DECL BOOL FraesAnford[10]
FraesAnford[1]=TRUE
FraesAnford[2]=TRUE
FraesAnford[3]=TRUE
FraesAnford[4]=FALSE
FraesAnford[5]=FALSE
FraesAnford[6]=FALSE
FraesAnford[7]=FALSE
FraesAnford[8]=FALSE
FraesAnford[9]=FALSE
FraesAnford[10]=FALSE
INT ERROR_PRG=0
;ENDFOLD
;FOLD USERSPOT_INPUTS_V4.xx
INT MAX_I_PS_MESSAGE=110
DECL I_MESSAGETYP PS_MESSAGE[110]
; EINGAENGE AM MODUL ZANGE 1
PS_MESSAGE[1]={I_NR 67,I_MSG_TXT[] "Stroemungswaechter Zange 1 E67 S42B                   "}
PS_MESSAGE[2]={I_NR 69,I_MSG_TXT[] "Vorhub Zange 1 hinten E69 B41YER                        "}
PS_MESSAGE[3]={I_NR 70,I_MSG_TXT[] "Schweisshub Zange 1 offen E70 B40YER                    "}
PS_MESSAGE[4]={I_NR 71,I_MSG_TXT[] "X-Vorhub Zange 1 vorne E71 B41YEV                       "}
PS_MESSAGE[5]={I_NR 72,I_MSG_TXT[] "Thermoschutz Trafo Zange 1 E72 B42TH                    "}
PS_MESSAGE[6]={I_NR 0,I_MSG_TXT[] " "}
PS_MESSAGE[7]={I_NR 0,I_MSG_TXT[] " "}
PS_MESSAGE[8]={I_NR 0,I_MSG_TXT[] " "}
PS_MESSAGE[9]={I_NR 0,I_MSG_TXT[] " "}

; EINGAENGE AM MODUL ZANGE 2
PS_MESSAGE[10]={I_NR 83,I_MSG_TXT[] "Stroemungswaechter Zange 2 E83 S12B                     "}
PS_MESSAGE[11]={I_NR 85,I_MSG_TXT[] "Vorhub Zange 2 hinten E85 B11YER                        "}
PS_MESSAGE[12]={I_NR 86,I_MSG_TXT[] "Schweisshub Zange 2 offen E86 B10YER                    "}
PS_MESSAGE[13]={I_NR 87,I_MSG_TXT[] "X-Vorhub Zange 2 vorne E87 B11YEV                       "}
PS_MESSAGE[14]={I_NR 88,I_MSG_TXT[] "Thermoschutz Trafo Zange 2 E88 B12TH                    "}
PS_MESSAGE[15]={I_NR 0,I_MSG_TXT[] " "}
PS_MESSAGE[16]={I_NR 0,I_MSG_TXT[] " "}
PS_MESSAGE[17]={I_NR 0,I_MSG_TXT[] " "}
PS_MESSAGE[18]={I_NR 0,I_MSG_TXT[] " "}


; EINGAENGE AM MODUL ZANGE 3
PS_MESSAGE[19]={I_NR 99,I_MSG_TXT[] "Stroemungswaechter Zange 3 E99 S22B                     "}
PS_MESSAGE[20]={I_NR 101,I_MSG_TXT[] "Vorhub Zange 3 hinten E101 B21YER                       "}
PS_MESSAGE[21]={I_NR 102,I_MSG_TXT[] "Schweisshub Zange 3 offen E102 B20YER                   "}
PS_MESSAGE[22]={I_NR 103,I_MSG_TXT[] "X-Vorhub Zange 3 vorne E103 B21YEV                      "}
PS_MESSAGE[23]={I_NR 104,I_MSG_TXT[] "Thermoschutz Trafo Zange 3 E104 B22TH                   "}
PS_MESSAGE[24]={I_NR 0,I_MSG_TXT[] " "}
PS_MESSAGE[25]={I_NR 0,I_MSG_TXT[] " "}
PS_MESSAGE[26]={I_NR 0,I_MSG_TXT[] " "}
PS_MESSAGE[27]={I_NR 0,I_MSG_TXT[] " "}



PS_MESSAGE[28]={I_NR 0,I_MSG_TXT[] "                            "}

PS_MESSAGE[29]={I_NR 817,I_MSG_TXT[] "Halt nach Applications Stop aktiv ! E817 HPE             "}

; Schweiss-Steuerung 1
PS_MESSAGE[30]={I_NR 225,I_MSG_TXT[] "FK E225 SWP1FK                                           "}
PS_MESSAGE[31]={I_NR 226,I_MSG_TXT[] "Anforderung Fraesen SWP1 E226 SWP1FR                      "}
PS_MESSAGE[32]={I_NR 227,I_MSG_TXT[] "Vorwarnung E227 SWP1WARN                                 "}
PS_MESSAGE[33]={I_NR 228,I_MSG_TXT[] "Maximale Standmenge erreicht E228 SWP1MAX                "}
PS_MESSAGE[34]={I_NR 229,I_MSG_TXT[] "ZPS bereit E229 SWP1BER                                  "}
PS_MESSAGE[35]={I_NR 230,I_MSG_TXT[] "Schweissfehler E230 SWP1SF                               "}
PS_MESSAGE[36]={I_NR 231,I_MSG_TXT[] "Schweissprozessueberwachung aus E231 SWP1UEWN            "}
PS_MESSAGE[37]={I_NR 232,I_MSG_TXT[] "Mit Schweissstrom E232 SWP1STR                           "}
PS_MESSAGE[38]={I_NR 0,I_MSG_TXT[] "Elektrode gewechselt/Startfraesen E234 SWP1STFR          "}
PS_MESSAGE[39]={I_NR 0,I_MSG_TXT[] "Neue Elektrode E235 SWP1NEEL                             "}
PS_MESSAGE[40]={I_NR 0,I_MSG_TXT[] "Fraesmesserverschleiss E236 SWP1FRVER                     "}
PS_MESSAGE[41]={I_NR 0,I_MSG_TXT[] "Fraesmesservorwarnung E237 SWP1FRWARN                     "}
PS_MESSAGE[42]={I_NR 0,I_MSG_TXT[] "Bauteil-End I247                                        "}
PS_MESSAGE[43]={I_NR 0,I_MSG_TXT[] "Punktanwahl gueltig I288                                 "}
PS_MESSAGE[44]={I_NR 0,I_MSG_TXT[] "                    "}
PS_MESSAGE[45]={I_NR 0,I_MSG_TXT[] "                    "}
PS_MESSAGE[46]={I_NR 0,I_MSG_TXT[] "                    "}
PS_MESSAGE[47]={I_NR 0,I_MSG_TXT[] "                    "}
PS_MESSAGE[48]={I_NR 0,I_MSG_TXT[] "                    "}
PS_MESSAGE[49]={I_NR 241,I_MSG_TXT[] "Motorschutz Fraesen SWP1 E241                    "}

; Schweiss-Steuerung 2
PS_MESSAGE[50]={I_NR 0,I_MSG_TXT[] "FK E257 SWP2FK                                           "}
PS_MESSAGE[51]={I_NR 0,I_MSG_TXT[] "Anforderung Fraesen SWP2 E258 SWP2FR                      "}
PS_MESSAGE[52]={I_NR 0,I_MSG_TXT[] "Vorwarnung E259 SWP2WARN                                 "}
PS_MESSAGE[53]={I_NR 0,I_MSG_TXT[] "Maximale Standmenge erreicht E260 SWP2MAX                "}
PS_MESSAGE[54]={I_NR 0,I_MSG_TXT[] "ZPS bereit E261 SWP2BER                                  "}
PS_MESSAGE[55]={I_NR 0,I_MSG_TXT[] "Schweissfehler E262 SWP2SF                               "}
PS_MESSAGE[56]={I_NR 0,I_MSG_TXT[] "Schweissprozessueberwachung aus E263 SWP2UEWN            "}
PS_MESSAGE[57]={I_NR 0,I_MSG_TXT[] "Mit Schweissstrom E264 SWP2STR                           "}
PS_MESSAGE[58]={I_NR 0,I_MSG_TXT[] "Elektrode gewechselt/Startfraesen E265 SWP2STFR          "}
PS_MESSAGE[59]={I_NR 0,I_MSG_TXT[] "Neue Elektrode E266 SWP2NEEL                             "}
PS_MESSAGE[60]={I_NR 0,I_MSG_TXT[] "Fraesmesserverschleiss E140 SWP1FRVER                     "}
PS_MESSAGE[61]={I_NR 0,I_MSG_TXT[] "Fraesmesservorwarnung E141 SWP1FRWARN                     "}
PS_MESSAGE[62]={I_NR 0,I_MSG_TXT[] "                    "}
PS_MESSAGE[63]={I_NR 0,I_MSG_TXT[] "                    "}
PS_MESSAGE[64]={I_NR 0,I_MSG_TXT[] "                    "}
PS_MESSAGE[65]={I_NR 0,I_MSG_TXT[] "                    "}
PS_MESSAGE[66]={I_NR 0,I_MSG_TXT[] "                    "}
PS_MESSAGE[67]={I_NR 0,I_MSG_TXT[] "                    "}
PS_MESSAGE[68]={I_NR 0,I_MSG_TXT[] "                    "}
PS_MESSAGE[69]={I_NR 0,I_MSG_TXT[] "Motorschutz Fraesen SWP2 E145                    "}

;Fräser 1
PS_MESSAGE[70]={I_NR 120,I_MSG_TXT[] "Fraeser 1 dreht E120 B46YM1                             "}
PS_MESSAGE[71]={I_NR 0,I_MSG_TXT[] "Fraesfertigmeldung 1 E143           "}
PS_MESSAGE[72]={I_NR 0,I_MSG_TXT[] "Fehler Fraesen 1 E144        "}
PS_MESSAGE[73]={I_NR 0,I_MSG_TXT[] "Kontrollsensor Fraesen 1 E147            "}
PS_MESSAGE[74]={I_NR 0,I_MSG_TXT[] "       "}

;Fräser 2
PS_MESSAGE[75]={I_NR 136,I_MSG_TXT[] "Fraeser 2 dreht E136 B16YM1                             "}
PS_MESSAGE[76]={I_NR 0,I_MSG_TXT[] "Fraesfertigmeldung 1 E143           "}
PS_MESSAGE[77]={I_NR 0,I_MSG_TXT[] "Fehler Fraesen 1 E144        "}
PS_MESSAGE[78]={I_NR 0,I_MSG_TXT[] "Kontrollsensor Fraesen 1 E147            "}
PS_MESSAGE[79]={I_NR 0,I_MSG_TXT[] "       "}

;Fräser 3
PS_MESSAGE[80]={I_NR 0,I_MSG_TXT[] "Fraeser 3 dreht E147 B26YM1                             "}
PS_MESSAGE[81]={I_NR 0,I_MSG_TXT[] "Fraesfertigmeldung 1 E143           "}
PS_MESSAGE[82]={I_NR 0,I_MSG_TXT[] "Fehler Fraesen 1 E144        "}
PS_MESSAGE[83]={I_NR 0,I_MSG_TXT[] "Kontrollsensor Fraesen 1 E147            "}
PS_MESSAGE[84]={I_NR 0,I_MSG_TXT[] "       "}

;Fräser 4
PS_MESSAGE[85]={I_NR 0,I_MSG_TXT[] "Fraeser 1 dreht E142       "}
PS_MESSAGE[86]={I_NR 0,I_MSG_TXT[] "Fraesfertigmeldung 1 E143           "}
PS_MESSAGE[87]={I_NR 0,I_MSG_TXT[] "Fehler Fraesen 1 E144        "}
PS_MESSAGE[88]={I_NR 0,I_MSG_TXT[] "Kontrollsensor Fraesen 1 E147            "}
PS_MESSAGE[89]={I_NR 0,I_MSG_TXT[] "       "}

;Schwenkeinheiten für Fräser
PS_MESSAGE[90]={I_NR 118,I_MSG_TXT[] "Schwenkeinrichtung vorn Fraeser1 E118 B45YEV            "}
PS_MESSAGE[91]={I_NR 134,I_MSG_TXT[] "Schwenkeinrichtung vorn Fraeser2 E134 B15YEV            "}
PS_MESSAGE[92]={I_NR 150,I_MSG_TXT[] "Schwenkeinrichtung vorn Fraeser3 E150 B25YEV            "}
PS_MESSAGE[93]={I_NR 116,I_MSG_TXT[] "Schwenkeinrichtung zurueck Fraeser1 E116  B45YER        "}
PS_MESSAGE[94]={I_NR 132,I_MSG_TXT[] "Schwenkeinrichtung zurueck Fraeser2 E132  B15YER        "}
PS_MESSAGE[95]={I_NR 148,I_MSG_TXT[] "Schwenkeinrichtung zurueck Fraeser3 E148  B25YER        "}
PS_MESSAGE[96]={I_NR 150,I_MSG_TXT[] "Schwenkeinrichtung zurueck Fraeser3 E516  B25YER        "}
PS_MESSAGE[97]={I_NR 0,I_MSG_TXT[] "Schwenkeinrichtung vorn Fraeser3 E153 B25YEV            "}
PS_MESSAGE[98]={I_NR 0,I_MSG_TXT[] " "}
PS_MESSAGE[99]={I_NR 0,I_MSG_TXT[] " "}

;Sonstiges
PS_MESSAGE[100]={I_NR 0,I_MSG_TXT[] " "}
PS_MESSAGE[101]={I_NR 0,I_MSG_TXT[] " "}
PS_MESSAGE[102]={I_NR 0,I_MSG_TXT[] " "}
PS_MESSAGE[103]={I_NR 0,I_MSG_TXT[] " "}
PS_MESSAGE[104]={I_NR 0,I_MSG_TXT[] " "}
PS_MESSAGE[105]={I_NR 0,I_MSG_TXT[] " "}
PS_MESSAGE[106]={I_NR 0,I_MSG_TXT[] " "}
PS_MESSAGE[107]={I_NR 0,I_MSG_TXT[] " "}
PS_MESSAGE[108]={I_NR 0,I_MSG_TXT[] " "}
PS_MESSAGE[109]={I_NR 0,I_MSG_TXT[] " "}
PS_MESSAGE[110]={I_NR 0,I_MSG_TXT[] "Kein Eingangsname definiert in Userspot.dat               "}


DECL I_MESSAGETYP PS_MESSAGE_U[110]
; EINGAENGE AM MODUL ZANGE 1
PS_MESSAGE_U[1]={I_NR 67,I_MSG_TXT[] "Stroemungswaechter Zange 1 E67 S42B                   "}
PS_MESSAGE_U[2]={I_NR 69,I_MSG_TXT[] "Vorhub Zange 1 hinten E69 B41YER                        "}
PS_MESSAGE_U[3]={I_NR 70,I_MSG_TXT[] "Schweisshub Zange 1 offen E70 B40YER                    "}
PS_MESSAGE_U[4]={I_NR 71,I_MSG_TXT[] "X-Vorhub Zange 1 vorne E71 B41YEV                       "}
PS_MESSAGE_U[5]={I_NR 72,I_MSG_TXT[] "Thermoschutz Trafo Zange 1 E72 B42TH                    "}
PS_MESSAGE_U[6]={I_NR 0,I_MSG_TXT[] " "}
PS_MESSAGE_U[7]={I_NR 0,I_MSG_TXT[] " "}
PS_MESSAGE_U[8]={I_NR 0,I_MSG_TXT[] " "}
PS_MESSAGE_U[9]={I_NR 0,I_MSG_TXT[] " "}

; EINGAENGE AM MODUL ZANGE 2
PS_MESSAGE_U[10]={I_NR 83,I_MSG_TXT[] "Stroemungswaechter Zange 2 E83 S12B                     "}
PS_MESSAGE_U[11]={I_NR 85,I_MSG_TXT[] "Vorhub Zange 2 hinten E85 B11YER                        "}
PS_MESSAGE_U[12]={I_NR 86,I_MSG_TXT[] "Schweisshub Zange 2 offen E86 B10YER                    "}
PS_MESSAGE_U[13]={I_NR 87,I_MSG_TXT[] "X-Vorhub Zange 2 vorne E87 B11YEV                       "}
PS_MESSAGE_U[14]={I_NR 88,I_MSG_TXT[] "Thermoschutz Trafo Zange 2 E88 B12TH                    "}
PS_MESSAGE_U[15]={I_NR 0,I_MSG_TXT[] " "}
PS_MESSAGE_U[16]={I_NR 0,I_MSG_TXT[] " "}
PS_MESSAGE_U[17]={I_NR 0,I_MSG_TXT[] " "}
PS_MESSAGE_U[18]={I_NR 0,I_MSG_TXT[] " "}


; EINGAENGE AM MODUL ZANGE 3
PS_MESSAGE_U[19]={I_NR 99,I_MSG_TXT[] "Stroemungswaechter Zange 3 E99 S22B                     "}
PS_MESSAGE_U[20]={I_NR 101,I_MSG_TXT[] "Vorhub Zange 3 hinten E101 B21YER                       "}
PS_MESSAGE_U[21]={I_NR 102,I_MSG_TXT[] "Schweisshub Zange 3 offen E102 B20YER                   "}
PS_MESSAGE_U[22]={I_NR 103,I_MSG_TXT[] "X-Vorhub Zange 3 vorne E103 B21YEV                      "}
PS_MESSAGE_U[23]={I_NR 104,I_MSG_TXT[] "Thermoschutz Trafo Zange 3 E104 B22TH                   "}
PS_MESSAGE_U[24]={I_NR 0,I_MSG_TXT[] " "}
PS_MESSAGE_U[25]={I_NR 0,I_MSG_TXT[] " "}
PS_MESSAGE_U[26]={I_NR 0,I_MSG_TXT[] " "}
PS_MESSAGE_U[27]={I_NR 0,I_MSG_TXT[] " "}



PS_MESSAGE_U[28]={I_NR 0,I_MSG_TXT[] "                            "}

PS_MESSAGE_U[29]={I_NR 817,I_MSG_TXT[] "Halt nach Applications Stop aktiv ! E817 HPE             "}

; Schweiss-Steuerung 1
PS_MESSAGE_U[30]={I_NR 225,I_MSG_TXT[] "FK E225 SWP1FK                                           "}
PS_MESSAGE_U[31]={I_NR 226,I_MSG_TXT[] "Anforderung Fraesen SWP1 E226 SWP1FR                      "}
PS_MESSAGE_U[32]={I_NR 227,I_MSG_TXT[] "Vorwarnung E227 SWP1WARN                                 "}
PS_MESSAGE_U[33]={I_NR 228,I_MSG_TXT[] "Maximale Standmenge erreicht E228 SWP1MAX                "}
PS_MESSAGE_U[34]={I_NR 229,I_MSG_TXT[] "ZPS bereit E229 SWP1BER                                  "}
PS_MESSAGE_U[35]={I_NR 230,I_MSG_TXT[] "Schweissfehler E230 SWP1SF                               "}
PS_MESSAGE_U[36]={I_NR 231,I_MSG_TXT[] "Schweissprozessueberwachung aus E231 SWP1UEWN            "}
PS_MESSAGE_U[37]={I_NR 232,I_MSG_TXT[] "Mit Schweissstrom E232 SWP1STR                           "}
PS_MESSAGE_U[38]={I_NR 0,I_MSG_TXT[] "Elektrode gewechselt/Startfraesen E234 SWP1STFR          "}
PS_MESSAGE_U[39]={I_NR 0,I_MSG_TXT[] "Neue Elektrode E235 SWP1NEEL                             "}
PS_MESSAGE_U[40]={I_NR 0,I_MSG_TXT[] "Fraesmesserverschleiss E236 SWP1FRVER                     "}
PS_MESSAGE_U[41]={I_NR 0,I_MSG_TXT[] "Fraesmesservorwarnung E237 SWP1FRWARN                     "}
PS_MESSAGE_U[42]={I_NR 0,I_MSG_TXT[] "Bauteil-End I247                                        "}
PS_MESSAGE_U[43]={I_NR 0,I_MSG_TXT[] "Punktanwahl gueltig I288                                 "}
PS_MESSAGE_U[44]={I_NR 0,I_MSG_TXT[] "                    "}
PS_MESSAGE_U[45]={I_NR 0,I_MSG_TXT[] "                    "}
PS_MESSAGE_U[46]={I_NR 0,I_MSG_TXT[] "                    "}
PS_MESSAGE_U[47]={I_NR 0,I_MSG_TXT[] "                    "}
PS_MESSAGE_U[48]={I_NR 0,I_MSG_TXT[] "                    "}
PS_MESSAGE_U[49]={I_NR 241,I_MSG_TXT[] "Motorschutz Fraesen SWP1 E241                    "}

; Schweiss-Steuerung 2
PS_MESSAGE_U[50]={I_NR 0,I_MSG_TXT[] "FK E257 SWP2FK                                           "}
PS_MESSAGE_U[51]={I_NR 0,I_MSG_TXT[] "Anforderung Fraesen SWP2 E258 SWP2FR                      "}
PS_MESSAGE_U[52]={I_NR 0,I_MSG_TXT[] "Vorwarnung E259 SWP2WARN                                 "}
PS_MESSAGE_U[53]={I_NR 0,I_MSG_TXT[] "Maximale Standmenge erreicht E260 SWP2MAX                "}
PS_MESSAGE_U[54]={I_NR 0,I_MSG_TXT[] "ZPS bereit E261 SWP2BER                                  "}
PS_MESSAGE_U[55]={I_NR 0,I_MSG_TXT[] "Schweissfehler E262 SWP2SF                               "}
PS_MESSAGE_U[56]={I_NR 0,I_MSG_TXT[] "Schweissprozessueberwachung aus E263 SWP2UEWN            "}
PS_MESSAGE_U[57]={I_NR 0,I_MSG_TXT[] "Mit Schweissstrom E264 SWP2STR                           "}
PS_MESSAGE_U[58]={I_NR 0,I_MSG_TXT[] "Elektrode gewechselt/Startfraesen E265 SWP2STFR          "}
PS_MESSAGE_U[59]={I_NR 0,I_MSG_TXT[] "Neue Elektrode E266 SWP2NEEL                             "}
PS_MESSAGE_U[60]={I_NR 0,I_MSG_TXT[] "Fraesmesserverschleiss E140 SWP1FRVER                     "}
PS_MESSAGE_U[61]={I_NR 0,I_MSG_TXT[] "Fraesmesservorwarnung E141 SWP1FRWARN                     "}
PS_MESSAGE_U[62]={I_NR 0,I_MSG_TXT[] "                    "}
PS_MESSAGE_U[63]={I_NR 0,I_MSG_TXT[] "                    "}
PS_MESSAGE_U[64]={I_NR 0,I_MSG_TXT[] "                    "}
PS_MESSAGE_U[65]={I_NR 0,I_MSG_TXT[] "                    "}
PS_MESSAGE_U[66]={I_NR 0,I_MSG_TXT[] "                    "}
PS_MESSAGE_U[67]={I_NR 0,I_MSG_TXT[] "                    "}
PS_MESSAGE_U[68]={I_NR 0,I_MSG_TXT[] "                    "}
PS_MESSAGE_U[69]={I_NR 0,I_MSG_TXT[] "Motorschutz Fraesen SWP2 E145                    "}

;Fräser 1
PS_MESSAGE_U[70]={I_NR 120,I_MSG_TXT[] "Fraeser 1 dreht E120 B46YM1                             "}
PS_MESSAGE_U[71]={I_NR 0,I_MSG_TXT[] "Fraesfertigmeldung 1 E143           "}
PS_MESSAGE_U[72]={I_NR 0,I_MSG_TXT[] "Fehler Fraesen 1 E144        "}
PS_MESSAGE_U[73]={I_NR 0,I_MSG_TXT[] "Kontrollsensor Fraesen 1 E147            "}
PS_MESSAGE_U[74]={I_NR 0,I_MSG_TXT[] "       "}

;Fräser 2
PS_MESSAGE_U[75]={I_NR 136,I_MSG_TXT[] "Fraeser 2 dreht E136 B16YM1                             "}
PS_MESSAGE_U[76]={I_NR 0,I_MSG_TXT[] "Fraesfertigmeldung 1 E143           "}
PS_MESSAGE_U[77]={I_NR 0,I_MSG_TXT[] "Fehler Fraesen 1 E144        "}
PS_MESSAGE_U[78]={I_NR 0,I_MSG_TXT[] "Kontrollsensor Fraesen 1 E147            "}
PS_MESSAGE_U[79]={I_NR 0,I_MSG_TXT[] "       "}

;Fräser 3
PS_MESSAGE_U[80]={I_NR 0,I_MSG_TXT[] "Fraeser 3 dreht E147 B26YM1                             "}
PS_MESSAGE_U[81]={I_NR 0,I_MSG_TXT[] "Fraesfertigmeldung 1 E143           "}
PS_MESSAGE_U[82]={I_NR 0,I_MSG_TXT[] "Fehler Fraesen 1 E144        "}
PS_MESSAGE_U[83]={I_NR 0,I_MSG_TXT[] "Kontrollsensor Fraesen 1 E147            "}
PS_MESSAGE_U[84]={I_NR 0,I_MSG_TXT[] "       "}

;Fräser 4
PS_MESSAGE_U[85]={I_NR 0,I_MSG_TXT[] "Fraeser 1 dreht E142       "}
PS_MESSAGE_U[86]={I_NR 0,I_MSG_TXT[] "Fraesfertigmeldung 1 E143           "}
PS_MESSAGE_U[87]={I_NR 0,I_MSG_TXT[] "Fehler Fraesen 1 E144        "}
PS_MESSAGE_U[88]={I_NR 0,I_MSG_TXT[] "Kontrollsensor Fraesen 1 E147            "}
PS_MESSAGE_U[89]={I_NR 0,I_MSG_TXT[] "       "}

;Schwenkeinheiten für Fräser
PS_MESSAGE_U[90]={I_NR 118,I_MSG_TXT[] "Schwenkeinrichtung vorn Fraeser1 E118 B45YEV            "}
PS_MESSAGE_U[91]={I_NR 134,I_MSG_TXT[] "Schwenkeinrichtung vorn Fraeser2 E134 B15YEV            "}
PS_MESSAGE_U[92]={I_NR 150,I_MSG_TXT[] "Schwenkeinrichtung vorn Fraeser3 E150 B25YEV            "}
PS_MESSAGE_U[93]={I_NR 116,I_MSG_TXT[] "Schwenkeinrichtung zurueck Fraeser1 E116  B45YER        "}
PS_MESSAGE_U[94]={I_NR 132,I_MSG_TXT[] "Schwenkeinrichtung zurueck Fraeser2 E132  B15YER        "}
PS_MESSAGE_U[95]={I_NR 148,I_MSG_TXT[] "Schwenkeinrichtung zurueck Fraeser3 E148  B25YER        "}
PS_MESSAGE_U[96]={I_NR 150,I_MSG_TXT[] "Schwenkeinrichtung zurueck Fraeser3 E516  B25YER        "}
PS_MESSAGE_U[97]={I_NR 0,I_MSG_TXT[] "Schwenkeinrichtung vorn Fraeser3 E153 B25YEV            "}
PS_MESSAGE_U[98]={I_NR 0,I_MSG_TXT[] " "}
PS_MESSAGE_U[99]={I_NR 0,I_MSG_TXT[] " "}

;Sonstiges
PS_MESSAGE_U[100]={I_NR 0,I_MSG_TXT[] " "}
PS_MESSAGE_U[101]={I_NR 0,I_MSG_TXT[] " "}
PS_MESSAGE_U[102]={I_NR 0,I_MSG_TXT[] " "}
PS_MESSAGE_U[103]={I_NR 0,I_MSG_TXT[] " "}
PS_MESSAGE_U[104]={I_NR 0,I_MSG_TXT[] " "}
PS_MESSAGE_U[105]={I_NR 0,I_MSG_TXT[] " "}
PS_MESSAGE_U[106]={I_NR 0,I_MSG_TXT[] " "}
PS_MESSAGE_U[107]={I_NR 0,I_MSG_TXT[] " "}
PS_MESSAGE_U[108]={I_NR 0,I_MSG_TXT[] " "}
PS_MESSAGE_U[109]={I_NR 0,I_MSG_TXT[] " "}
PS_MESSAGE_U[110]={I_NR 0,I_MSG_TXT[] "Kein Eingangsname definiert in Userspot.dat               "}


INT MAX_I_PS_MESSAGE1=4
DECL I_MESSAGETYP PS_MESSAGE1[10]
; EINGAENGE Twin-Fraeser
PS_MESSAGE1[1]={I_NR 0,I_MSG_TXT[] "Twin Fraeser 1 dreht E? B46YM2                        "}
PS_MESSAGE1[2]={I_NR 0,I_MSG_TXT[] "Twin Fraeser 2 dreht E? B16YM2                        "}
PS_MESSAGE1[3]={I_NR 0,I_MSG_TXT[] "Twin Fraeser 3 dreht E? B26YM2                        "}
PS_MESSAGE1[4]={I_NR 0,I_MSG_TXT[] "Kein Eingangsname vorhanden       "}

DECL I_MESSAGETYP PS_MESSAGE1_U[10]
; EINGAENGE Twin-Fraeser
PS_MESSAGE1_U[1]={I_NR 0,I_MSG_TXT[] "Twin Fraeser 1 dreht E? B46YM2                        "}
PS_MESSAGE1_U[2]={I_NR 0,I_MSG_TXT[] "Twin Fraeser 2 dreht E? B16YM2                        "}
PS_MESSAGE1_U[3]={I_NR 0,I_MSG_TXT[] "Twin Fraeser 3 dreht E? B26YM2                        "}
PS_MESSAGE1_U[4]={I_NR 0,I_MSG_TXT[] "Kein Eingangsname vorhanden       "}



;ENDFOLD
;FOLD USERSPOT_ERRORS_V4.xx
INT MAX_I_PS_ERROR=20
DECL MSG_TXT_TYP PS_ERROR[20]
PS_ERROR[1]={MSGTXT[] "Fraeser klemmt Fraesvorgang beenden ?  "}
PS_ERROR[2]={MSGTXT[] "Ungueltige Schweisskofferparametrierung !  "}
PS_ERROR[3]={MSGTXT[] "Zangenzahl oder Endschalter Ablage n.i.O   "}
PS_ERROR[4]={MSGTXT[] "Schweissueberw. ist ausgeschalten !           "}
PS_ERROR[5]={MSGTXT[] "Schweissstrom ist ausgeschaltet!  Einschalten ?  "}
PS_ERROR[6]={MSGTXT[] "Projektierungsfehler Fraeserzuordnung"}
PS_ERROR[7]={MSGTXT[] "GUN Nr. nicht in Userspot.dat (Zange[Gun]) definiert "}
PS_ERROR[8]={MSGTXT[] "Roboter gestoppt wegen fehlendem FK! Beheben und neu starten"}
PS_ERROR[9]={MSGTXT[] "FK von Schweisssteuerung fehlt!   Schweisssung wiederholen ?"}
PS_ERROR[10]={MSGTXT[] "! Konfiguration Fraeser nicht moeglich !"}
PS_ERROR[11]={MSGTXT[] " Abbruch, Fraespr. angewaehlt ! "}
PS_ERROR[12]={MSGTXT[] " Maximale Fraeserlaufzeit erreicht ! "}
PS_ERROR[13]={MSGTXT[] " Abruch Fraeser nicht gestartet ! "}
PS_ERROR[14]={MSGTXT[] " Abbruch !! Kein Fraeser parametriert !"}
PS_ERROR[15]={MSGTXT[] " Fraesfehler von der Schweisssteuerung !"}
PS_ERROR[16]={MSGTXT[] " Elektrode-Kontrolle ist nicht in Ordnung ! "}
PS_ERROR[17]={MSGTXT[] "Falsche Zange angedockt !                   "}
PS_ERROR[18]={MSGTXT[] " "}
PS_ERROR[19]={MSGTXT[] " "}
PS_ERROR[20]={MSGTXT[] " "}

DECL MSG_TXT_TYP PS_ERROR_U[20]
PS_ERROR_U[1]={MSGTXT[] "Fraeser klemmt Fraesvorgang beenden ?  "}
PS_ERROR_U[2]={MSGTXT[] "Ungueltige Schweisskofferparametrierung !  "}
PS_ERROR_U[3]={MSGTXT[] "Zangenzahl oder Endschalter Ablage n.i.O   "}
PS_ERROR_U[4]={MSGTXT[] "Schweissueberw. ist ausgeschalten !           "}
PS_ERROR_U[5]={MSGTXT[] "Schweissstrom ist ausgeschaltet!  Einschalten ?  "}
PS_ERROR_U[6]={MSGTXT[] "Projektierungsfehler Fraeserzuordnung"}
PS_ERROR_U[7]={MSGTXT[] "GUN Nr. nicht in Userspot.dat (Zange[Gun]) definiert "}
PS_ERROR_U[8]={MSGTXT[] "Roboter gestoppt wegen fehlendem FK! Beheben und neu starten"}
PS_ERROR_U[9]={MSGTXT[] "FK von Schweisssteuerung fehlt!   Schweisssung wiederholen ?"}
PS_ERROR_U[10]={MSGTXT[] "! Konfiguration Fraeser nicht moeglich !"}
PS_ERROR_U[11]={MSGTXT[] " Abbruch, Fraespr. angewaehlt ! "}
PS_ERROR_U[12]={MSGTXT[] " Maximale Fraeserlaufzeit erreicht ! "}
PS_ERROR_U[13]={MSGTXT[] " Abruch Fraeser nicht gestartet ! "}
PS_ERROR_U[14]={MSGTXT[] " Abbruch !! Kein Fraeser parametriert !"}
PS_ERROR_U[15]={MSGTXT[] " Fraesfehler von der Schweisssteuerung !"}
PS_ERROR_U[16]={MSGTXT[] " Elektrode-Kontrolle ist nicht in Ordnung ! "}
PS_ERROR_U[17]={MSGTXT[] "Falsche Zange angedockt !                   "}
PS_ERROR_U[18]={MSGTXT[] " "}
PS_ERROR_U[19]={MSGTXT[] " "}
PS_ERROR_U[20]={MSGTXT[] " "}

;ENDFOLD
;Fold Bosch Error Code V1.0
;Status-Codes vom Schweisskoffer auswerten
SIGNAL PS_SK_StatusIn $IN[257]  TO $IN[272]
STRUC PS_SK_SatusCodeTyp INT Nr,CHAR MsgText[50]
DECL INT PS_SK_SatusCodeMax=34
DECL PS_SK_SatusCodeTyp PS_SK_SatusCode[34]
PS_SK_SatusCode[1]={Nr 0,MsgText[] "Kein FK (IN%%1): %s, Wiederholung?"}
PS_SK_SatusCode[2]={Nr 0,MsgText[] "Schweissfehler(IN%%1): %s, Wiederholen?"}
PS_SK_SatusCode[3]={Nr 80,MsgText[] "Stopp Kreis offen / +24V fehlt         "}
PS_SK_SatusCode[4]={Nr 81,MsgText[] "SOB: Strom ohne Befehl                 "}
PS_SK_SatusCode[5]={Nr 84,MsgText[] "Batterie Fehler                        "}
PS_SK_SatusCode[6]={Nr 85,MsgText[] "Speicher geloescht==RAM Checksum Fehler"}
PS_SK_SatusCode[7]={Nr 86,MsgText[] "Daten - Restore aktiv                  "}
PS_SK_SatusCode[8]={Nr 87,MsgText[] "kein Schweissprogramm==ungueltige Param"}
PS_SK_SatusCode[9]={Nr 88,MsgText[] "Hardware Fehler                        "}
PS_SK_SatusCode[10]={Nr 89,MsgText[] "E/A Bus-Fehler                         "}
PS_SK_SatusCode[11]={Nr 90,MsgText[] "Halbwellen Ueberwachung                "}
PS_SK_SatusCode[12]={Nr 91,MsgText[] "Hauptschalter ausgeloest               "}
PS_SK_SatusCode[13]={Nr 92,MsgText[] "Externe Temperatur zu hoch             "}
PS_SK_SatusCode[14]={Nr 93,MsgText[] "Synchronisations-Fehler                "}
PS_SK_SatusCode[15]={Nr 94,MsgText[] "Ablauf gesperrt                        "}
PS_SK_SatusCode[16]={Nr 95,MsgText[] "Programm-Paritaet Fehler               "}
PS_SK_SatusCode[17]={Nr 98,MsgText[] "Sollwert zu Gross                      "}
PS_SK_SatusCode[18]={Nr 99,MsgText[] "Schweissprozess-Fehler                 "}
PS_SK_SatusCode[19]={Nr 100,MsgText[] "Versorgungsspannungs Fehler            "}
PS_SK_SatusCode[20]={Nr 160,MsgText[] "Kuehlkoerpertemperatur zu hoch         "}
PS_SK_SatusCode[21]={Nr 164,MsgText[] "Trafotemperatur zu hoch                "}
PS_SK_SatusCode[22]={Nr 165,MsgText[] "Hardwarefehler Treiberbaugruppe        "}
PS_SK_SatusCode[23]={Nr 166,MsgText[] "24V Versorgungsspannungsfehler         "}
PS_SK_SatusCode[24]={Nr 182,MsgText[] "Fraeseransteuerung fehlerhaft          "}
PS_SK_SatusCode[25]={Nr 224,MsgText[] "Fraeserg fehlerhaft bei erster Pruefung"}
PS_SK_SatusCode[26]={Nr 225,MsgText[] "Fraeserg fehlerhaft bei zweiter Pruefng"}
PS_SK_SatusCode[27]={Nr 3106,MsgText[] "Q-Stopp Bauteil                ------ "}
PS_SK_SatusCode[28]={Nr 3107,MsgText[] "Q-Stopp Punkt in Folge         ------ "}
PS_SK_SatusCode[29]={Nr 3108,MsgText[] "Q-Stopp Sonderpunkt            ------ "}
PS_SK_SatusCode[30]={Nr 3109,MsgText[] "Q-Stopp UIP absolut unten      ------ "}
PS_SK_SatusCode[31]={Nr 3110,MsgText[] "Q-Stopp PSF absolut unten      ------ "}
PS_SK_SatusCode[32]={Nr 3111,MsgText[] "Q-Stopp UIP absolut oben       ------ "}
PS_SK_SatusCode[33]={Nr 3112,MsgText[] "Q-Stopp FQF absolut unten      ------ "}
PS_SK_SatusCode[34]={Nr 3113,MsgText[] "Q-Stopp FQF absolut oben       ------ "}
;endfold (ErrorCode)
ENDDAT
